FUNCTION_BLOCK WaterMonitor_FBDKTestBench (* Composite Function Block Type *)
  (* Standard: 61499-2 *)
  (* Version 0.2, 2003-12-05, JHC, Rockwell Automation, Renamed from NEWCOMPFB. *)
  (* Version 0.1, 2002-01-08, JHC, Rockwell Automation, Added DLY FB as example. *)
  (* Version 0.0, 2000-05-27, JHC, Rockwell Automation *)
  (* Compiler header: package fb.rt.benchmarks.watermonitor; *)
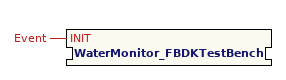
  EVENT_INPUT
    INIT; (* Initialization Request *)
  END_EVENT
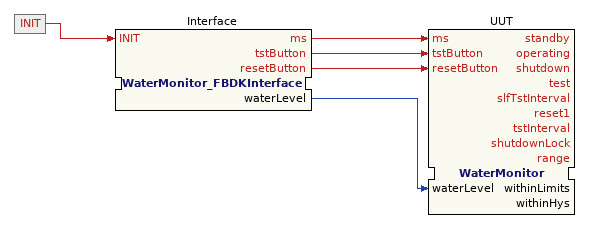
  FBS
    Interface : WaterMonitor_FBDKInterface;
    UUT : WaterMonitor;
  END_FBS
  EVENT_CONNECTIONS
    INIT TO Interface.INIT;
    Interface.ms TO UUT.ms;
    Interface.tstButton TO UUT.tstButton;
    Interface.resetButton TO UUT.resetButton;
  END_CONNECTIONS
  DATA_CONNECTIONS
    Interface.waterLevel TO UUT.waterLevel;
  END_CONNECTIONS
END_FUNCTION_BLOCK
